{attribute 'TcGenerated'}
{attribute 'no-analysis'}
{attribute 'linkalways'}
// This function has been automatically generated from the project information.
VAR_GLOBAL CONSTANT
	{attribute 'const_non_replaced'}
	stLibVersion_tcl_BaseClasses : ST_LibVersion := (iMajor := 1, iMinor := 1, iBuild := 31, iRevision := 0, nFlags := 0, sVersion := '1.1.31.0');
END_VAR

(* stored: Version 1.1.0.1, ProductVersion 3.1.4024.12
   GVL Global_Version: Id {69e73143-71b5-4371-b308-9ebb3c3f0c7f} *)
